(* LS Electric XG5000 project: Study5_sth_to_sth *)
(* PLC LSPLC *)

PROGRAM NewProgram (* task: 스캔 프로그램 *)
VAR
    input1 : REAL;
    output1 : INT;
END_VAR

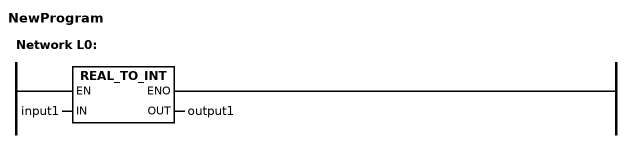
(* Rung L0 *)
output1 := REAL_TO_INT(input1);
END_PROGRAM